{attribute addProperty BoxType "EL3151-0000-0016"}
{attribute addProperty Id "AI_StandardAT %I*AI_Standard_8749C235749.250WcStateAT %I*WcState_F855686C1620InfoDataAT %I*InfoData_BC63D37F80100"}
{attribute addProperty CRC "2074988543"}
{attribute addProperty SizeInBites "170"}
{attribute addProperty SizeInBytes "21.25"}
TYPE EL3151_50D9316A :
STRUCT
	{attribute addProperty Name "AI_Standard"}
	AI_Standard : AI_Standard_8749C235;
	{attribute addProperty Name "WcState"}
	WcState : WcState_F855686C;
	{attribute addProperty Name "InfoData"}
	InfoData : InfoData_BC63D37F;
END_STRUCT
END_TYPE

(* stored: Version 1.2.0.0, ProductVersion 3.1.4024.9
   DUT EL3151_50D9316A: Id {344c6221-c144-4741-9796-d92d9a3558d7} *)
